Staubli VAL3: getPointData.pgx

program getPointData(num& x_nSpeed[], mdesc& x_mDesc[], num& x_nDistance[], bool& x_bToStop[], num& x_nMoveType[], num& x_nStop[], num x_nIndex, bool x_bCycle)
begin
  if x_bCycle
    // get tha parameter
    // SPEED
    // get the speed in mm/sec
    if pt:tTraj[sTrajCycle].tData[x_nIndex].tSuper.moveType==0
      x_nSpeed=pt:tTraj[sTrajCycle].tData[x_nIndex].tSuper.nom_speed.vel*15
    else
      if pt:tTraj[sTrajCycle].tData[x_nIndex].tSuper.moveType==1
        x_nSpeed=pt:tTraj[sTrajCycle].tData[x_nIndex].tSuper.nom_speed.tvel
      endIf
    endIf
    // MDESC
    x_mDesc=pt:tTraj[sTrajCycle].tData[x_nIndex].tSuper.nom_speed
    // DISTANCE
    x_nDistance=pt:tTraj[sTrajCycle].tData[x_nIndex].tSuper.distance
    //  check  for a stop using
    x_bToStop=pt:tTraj[sTrajCycle].tData[x_nIndex].tSuper.toStop
    // get MoveType
    x_nMoveType=pt:tTraj[sTrajCycle].tData[x_nIndex].tSuper.moveType
  else
    // get tha parameter
    // SPEED
    // get the speed in mm/sec
    if jEditPoint.tData[x_nIndex].tSuper.moveType==0
      x_nSpeed=jEditPoint.tData[x_nIndex].tSuper.nom_speed.vel*15
    else
      if jEditPoint.tData[x_nIndex].tSuper.moveType==1
        x_nSpeed=jEditPoint.tData[x_nIndex].tSuper.nom_speed.tvel
      endIf
    endIf
    // MDESC
    x_mDesc=jEditPoint.tData[x_nIndex].tSuper.nom_speed
    // DISTANCE
    x_nDistance=jEditPoint.tData[x_nIndex].tSuper.distance
    //  check  for a stop using
    x_bToStop=jEditPoint.tData[x_nIndex].tSuper.toStop
    // get MoveType
    x_nMoveType=jEditPoint.tData[x_nIndex].tSuper.moveType
  endIf
end
